// TIA Portal V16 export
// export: Created 2021-07-12T14:47:20.6953747Z, ExportSetting WithDefaults, DisplayName Totally Integrated Automation Portal, DisplayVersion V16, DisplayName TIA Portal Version Control Interface, DisplayVersion V16, DisplayName TIA Portal Openness, DisplayVersion V16, DisplayName STEP 7 Professional, DisplayVersion V16, DisplayName STEP 7 Safety, DisplayVersion V16, DisplayName WinCC Professional, DisplayVersion V16
TYPE "SimaHydTO_typeHMIConnectionAxisToData"
TITLE = SimaHydTO_typeHMIConnectionAxisToData
// HMI interface: Technology object axis diagnostic words
// stored: IsFailsafeCompliant false
   STRUCT
      statusWord : DWord;
      warningWord : DWord;
      errorWord : DWord;
      errorDetail { S7_SetPoint := 'True'} : "SimaHydTO_typeHMIConnectionAxisToDataErrorDetail";
      axisUnits { S7_SetPoint := 'True'} : "SimaHydTO_typeHMIConnectionAxisToDataAxisUnits";
      typeOfAxis : Int;   // 0: No axis / 1: Speed axis / 2: Positioning axis / 3: Synchronous axis / 4: External encoder
   END_STRUCT;
END_TYPE
